(* Logix 5000 project; controller cal1615 1756-L62 rev 16.20; software revision 16.05; part 42 of 78 *)
(* tags used below, declared in another part *)
   AFI : BOOL;   // Always False Bit
   FAULT : BOOL;   // Fault AFI
   p01r02_plc_scan_time_in_sec : REAL;   // System PLC Scan Time in Seconds
   p01r09_pb_global_reset : BOOL;   // System Modes PB: Global Fault Reset
   p20_ao_lo_turret_selected_speed : REAL;   // Letoff Letoff Turret VFD Selected Speed
   p20_di_clutch_prs_ok : BOOL;   // Letoff Modes Accumulator Position Mode
   p20_di_lo_turret : acs800_di_normal;   // Letoff Letoff Turret VFD Drive Inputs
   p20_di_lo_turret_therm : BOOL;   // Letoff Input Letoff Turret Motor Temp Ok
   p20_di_turret_fwd : BOOL;   // Letoff Digital Inputs PB: Turret FWD
   p20_di_turret_pos : BOOL;   // Letoff Digital Inputs PX: Turret in Position
   p20_di_turret_rev : BOOL;   // Letoff Digital Inputs PB: Turret REV
   p20_do_close_nip : BOOL;   // Letoff Digital Output Feedroll Roll Nip Close
   p20_do_wdr_turret : acs800_do_normal;
   p20_param_lo_turret_index_speed : REAL;
   p20_request_run_index_dir : BOOL;   // Letoff Letoff Turret Request Run Index Direction
   p20_request_run_index_rev_dir : BOOL;   // Letoff Letoff Turret Request Run Index Reverse Direction
   p20r01 : routine;   // Letoff Main
   p20r15 : routine;   // Letoff Letoff A VFD
   p20r15_loa_on : BOOL;   // Letoff Letoff A VFD On
   p20r16_lob_on : BOOL;   // Letoff Letoff B On
   p20r18 : routine;   // Letoff Letoff Turret VFD
   p20r18_acc_dec_ramp : SYS_ACC_DEC_RAMP;   // Letoff Letoff Turret VFD Acel Decel Ramp
   p20r18_accel_rate : REAL;
   p20r18_decel_rate : REAL;
   p20r18_index_complete : BOOL;   // Letoff Letoff Turret VFD Index Complete
   p20r18_index_move_timer : TIMER;   // Letoff Letoff Turret VFD Move Timer
   p20r18_index_time : DINT;   // Letoff Letoff Turret Index Time
   p20r18_index_time_offset : DINT;   // Letoff Letoff Turret VFD Index Time Offset (Accel/Decel Rate Difference)
   p20r18_index_timer : TIMER;   // Letoff Letoff Turret Index Timer
   p20r18_pb_index_fwd : BOOL;   // Letoff Letoff Turret VFD PB: Index FWD
   p20r18_pb_index_rev : BOOL;   // Letoff Letoff Turret VFD PB: Index REV
   p20r18_permissive : BOOL;   // Letoff Letoff Turret VFD Permissive
   p20r18_request_index_fwd : BOOL;   // Letoff Letoff Turret Request Index Forward
   p20r18_request_index_rev : BOOL;   // Letoff Letoff Turret Request Index Reverse
   p20r18_selected_speed : REAL;   // Letoff Letoff Turret VFD Selected Speed
   p20r18_timer_fault : TIMER[10];   // Letoff Letoff Turret Fault Dwell Timer
   p20r18_timer_warning : TIMER[4];   // Letoff Letoff Turret VFD Warning Dwell Timer
   p20r18_zero_speed : BOOL;   // Letoff Letoff Turret VFD At Zero Speed
   p21_dint_to_hmi : DINT[16];   // Splice Press
   P21r01 : routine;
   p21r02 : routine;   // Splice Press Misc Control
   p21r02_fault_exists : BOOL;
   p21r02_timer_fault : TIMER[4];   // Splice Press Misc Control Fault Delay
   p21r02_timer_warning : TIMER[4];   // Splice Press Misc Control Warning Delay
   p21r02_unack_fault : BOOL;   // Splice Press Misc Control Unacknowledged Fault Exists
   p21r02_unack_warning : BOOL;   // Splice Press Misc Control Unacknowledged Warning Exists
   p21r02_warning_exists : BOOL;
   p21r03 : routine;   // Splice Press Inputs
   p21r04 : routine;   // Splice Press Outputs
   p21r05 : routine;   // Splice Press Dint to HMI
   p21r06 : routine;   // Splice Press Real to HMI
   p21r07 : routine;   // Splice Press Alarms
   p21r08 : routine;   // Splice Press Warnings
   p21r09 : routine;   // Splice Press Modes
   p21r10 : routine;   // Splice Press Sequence
   p21r16 : routine;   // Splice Press Temperature Control
(* P20_Letoff, continued *)

ROUTINE R18_Letoff_Turret_VFD   (* ladder *)
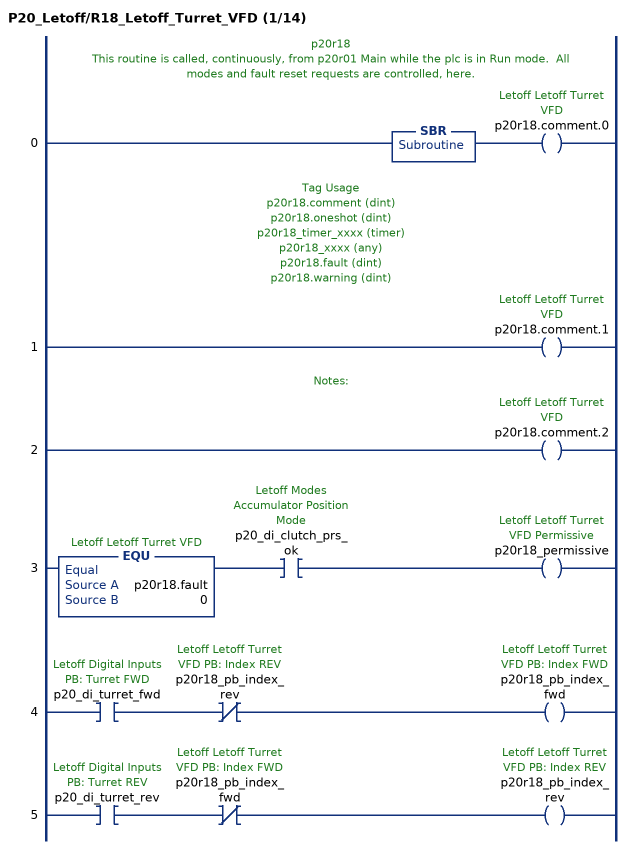
   // p20r18
   // This routine is called, continuously, from p20r01 Main while the plc is in Run mode.  All modes and fault reset requests are controlled, here.
   0: SBR()OTE(p20r18.comment.0);
   // Tag Usage
   // p20r18.comment (dint)
   // p20r18.oneshot (dint)
   // p20r18_timer_xxxx (timer)
   // p20r18_xxxx (any)
   // p20r18.fault (dint)
   // p20r18.warning (dint)
   1: OTE(p20r18.comment.1);
   // Notes:
   2: OTE(p20r18.comment.2);
   3: EQU(p20r18.fault,0)XIC(p20_di_clutch_prs_ok)OTE(p20r18_permissive);
   4: XIC(p20_di_turret_fwd)XIO(p20r18_pb_index_rev)OTE(p20r18_pb_index_fwd);
   5: XIC(p20_di_turret_rev)XIO(p20r18_pb_index_fwd)OTE(p20r18_pb_index_rev);
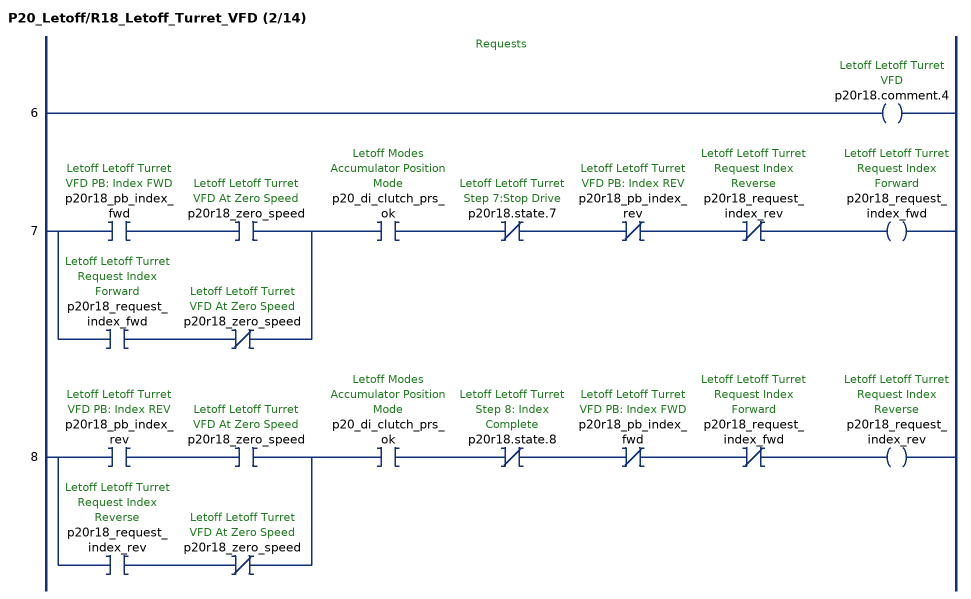
   // Requests
   6: OTE(p20r18.comment.4);
   7: [XIC(p20r18_pb_index_fwd) XIC(p20r18_zero_speed) ,XIC(p20r18_request_index_fwd) XIO(p20r18_zero_speed) ]XIC(p20_di_clutch_prs_ok)XIO(p20r18.state.7)XIO(p20r18_pb_index_rev)XIO(p20r18_request_index_rev)OTE(p20r18_request_index_fwd);
   8: [XIC(p20r18_pb_index_rev) XIC(p20r18_zero_speed) ,XIC(p20r18_request_index_rev) XIO(p20r18_zero_speed) ]XIC(p20_di_clutch_prs_ok)XIO(p20r18.state.8)XIO(p20r18_pb_index_fwd)XIO(p20r18_request_index_fwd)OTE(p20r18_request_index_rev);
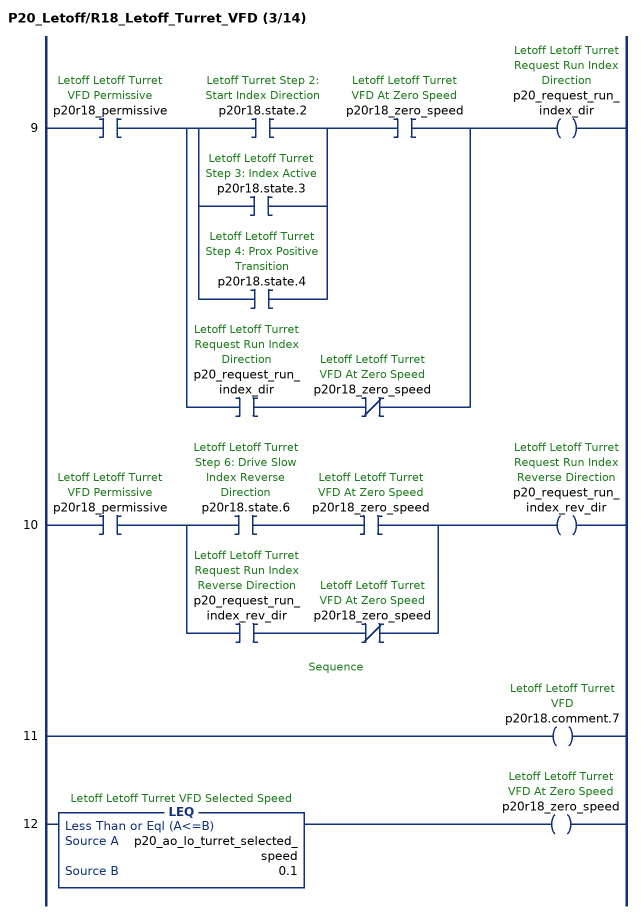
   9: XIC(p20r18_permissive)[[XIC(p20r18.state.2) ,XIC(p20r18.state.3) ,XIC(p20r18.state.4) ] XIC(p20r18_zero_speed) ,XIC(p20_request_run_index_dir) XIO(p20r18_zero_speed) ]OTE(p20_request_run_index_dir);
   10: XIC(p20r18_permissive)[XIC(p20r18.state.6) XIC(p20r18_zero_speed) ,XIC(p20_request_run_index_rev_dir) XIO(p20r18_zero_speed) ]OTE(p20_request_run_index_rev_dir);
   // Sequence
   11: OTE(p20r18.comment.7);
   12: LEQ(p20_ao_lo_turret_selected_speed,0.1)OTE(p20r18_zero_speed);
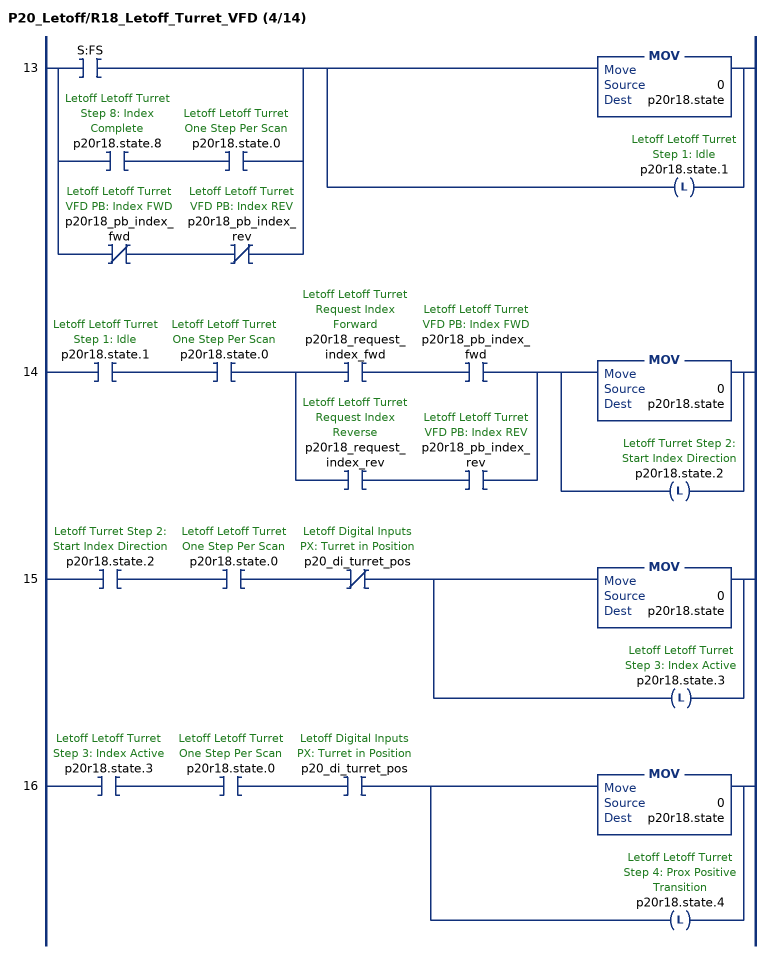
   13: [XIC(S:FS) ,XIC(p20r18.state.8) XIC(p20r18.state.0) ,XIO(p20r18_pb_index_fwd) XIO(p20r18_pb_index_rev) ][MOV(0,p20r18.state) ,OTL(p20r18.state.1) ];
   14: XIC(p20r18.state.1)XIC(p20r18.state.0)[XIC(p20r18_request_index_fwd) XIC(p20r18_pb_index_fwd) ,XIC(p20r18_request_index_rev) XIC(p20r18_pb_index_rev) ][MOV(0,p20r18.state) ,OTL(p20r18.state.2) ];
   15: XIC(p20r18.state.2)XIC(p20r18.state.0)XIO(p20_di_turret_pos)[MOV(0,p20r18.state) ,OTL(p20r18.state.3) ];
   16: XIC(p20r18.state.3)XIC(p20r18.state.0)XIC(p20_di_turret_pos)[MOV(0,p20r18.state) ,OTL(p20r18.state.4) ];
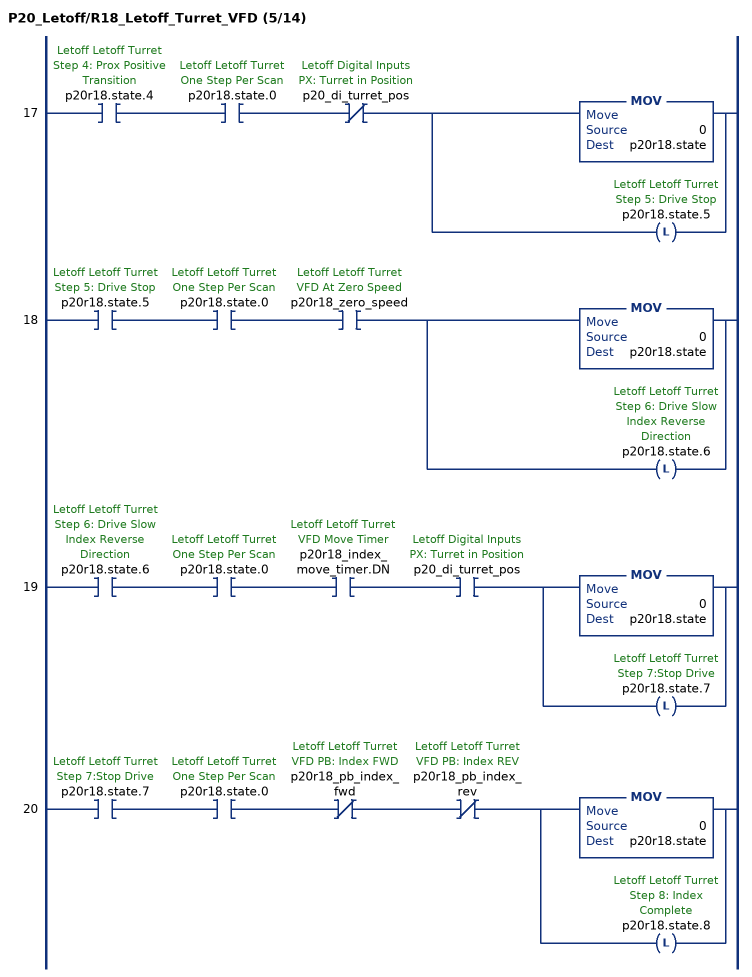
   17: XIC(p20r18.state.4)XIC(p20r18.state.0)XIO(p20_di_turret_pos)[MOV(0,p20r18.state) ,OTL(p20r18.state.5) ];
   18: XIC(p20r18.state.5)XIC(p20r18.state.0)XIC(p20r18_zero_speed)[MOV(0,p20r18.state) ,OTL(p20r18.state.6) ];
   19: XIC(p20r18.state.6)XIC(p20r18.state.0)XIC(p20r18_index_move_timer.DN)XIC(p20_di_turret_pos)[MOV(0,p20r18.state) ,OTL(p20r18.state.7) ];
   20: XIC(p20r18.state.7)XIC(p20r18.state.0)XIO(p20r18_pb_index_fwd)XIO(p20r18_pb_index_rev)[MOV(0,p20r18.state) ,OTL(p20r18.state.8) ];
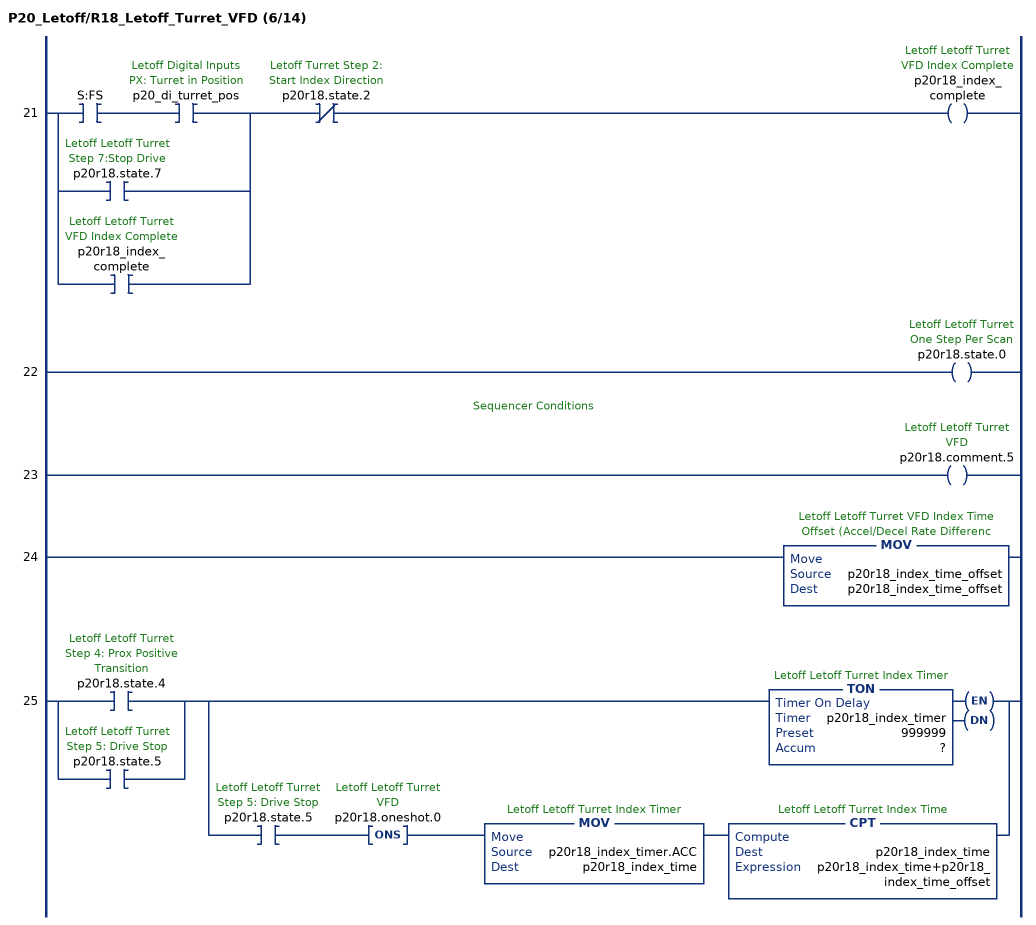
   21: [XIC(S:FS) XIC(p20_di_turret_pos) ,XIC(p20r18.state.7) ,XIC(p20r18_index_complete) ]XIO(p20r18.state.2)OTE(p20r18_index_complete);
   22: OTE(p20r18.state.0);
   // Sequencer Conditions
   23: OTE(p20r18.comment.5);
   24: MOV(p20r18_index_time_offset,p20r18_index_time_offset);
   25: [XIC(p20r18.state.4) ,XIC(p20r18.state.5) ][TON(p20r18_index_timer,?,?) ,XIC(p20r18.state.5) ONS(p20r18.oneshot.0) MOV(p20r18_index_timer.ACC,p20r18_index_time) CPT(p20r18_index_time,p20r18_index_time+p20r18_index_time_offset) ];
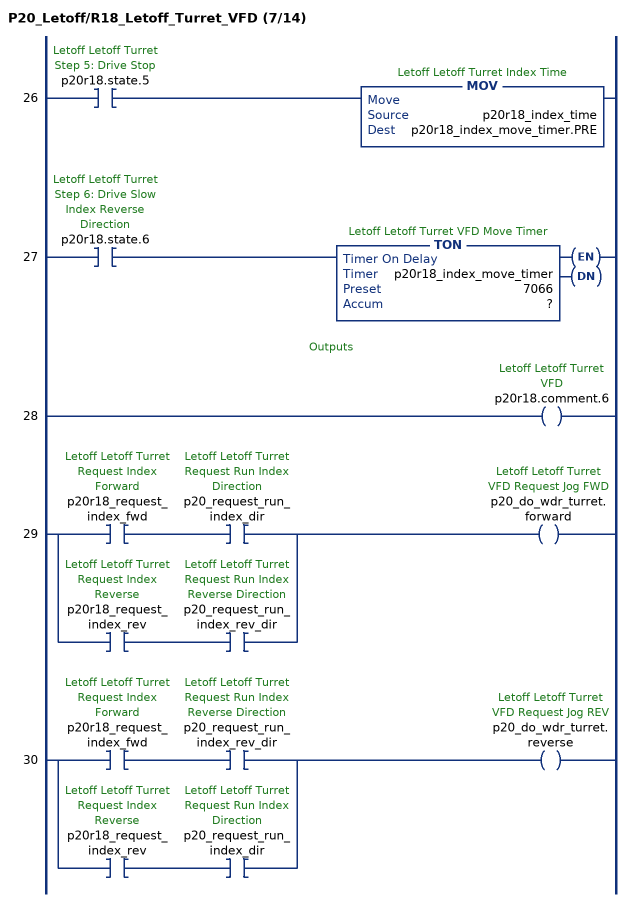
   26: XIC(p20r18.state.5)MOV(p20r18_index_time,p20r18_index_move_timer.PRE);
   27: XIC(p20r18.state.6)TON(p20r18_index_move_timer,?,?);
   // Outputs
   28: OTE(p20r18.comment.6);
   29: [XIC(p20r18_request_index_fwd) XIC(p20_request_run_index_dir) ,XIC(p20r18_request_index_rev) XIC(p20_request_run_index_rev_dir) ]OTE(p20_do_wdr_turret.forward);
   30: [XIC(p20r18_request_index_fwd) XIC(p20_request_run_index_rev_dir) ,XIC(p20r18_request_index_rev) XIC(p20_request_run_index_dir) ]OTE(p20_do_wdr_turret.reverse);
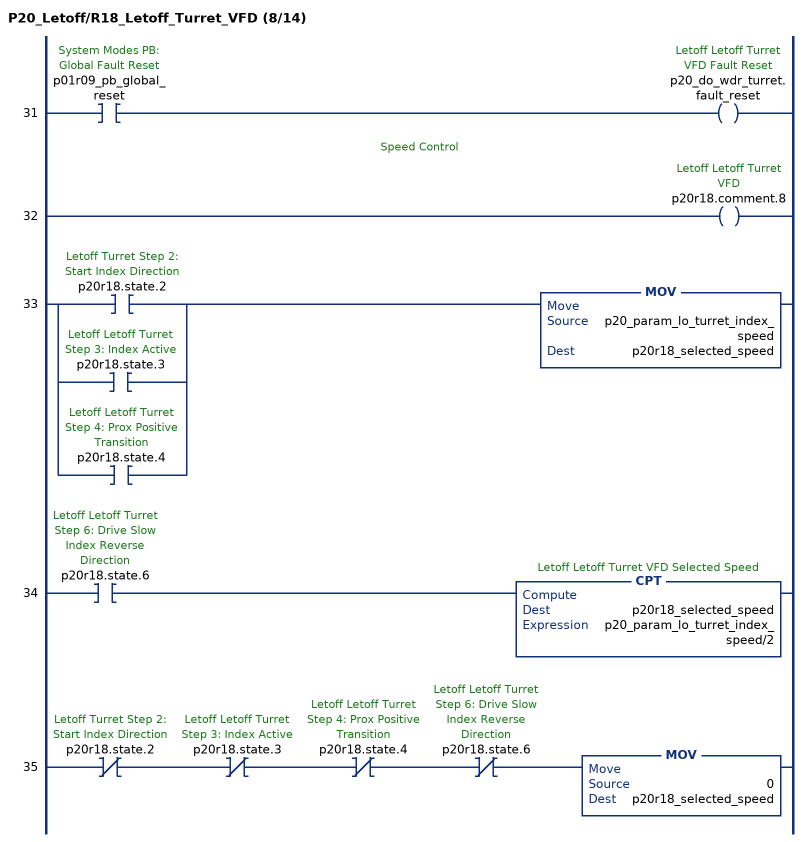
   31: XIC(p01r09_pb_global_reset)OTE(p20_do_wdr_turret.fault_reset);
   // Speed Control
   32: OTE(p20r18.comment.8);
   33: [XIC(p20r18.state.2) ,XIC(p20r18.state.3) ,XIC(p20r18.state.4) ]MOV(p20_param_lo_turret_index_speed,p20r18_selected_speed);
   34: XIC(p20r18.state.6)CPT(p20r18_selected_speed,p20_param_lo_turret_index_speed/2);
   35: XIO(p20r18.state.2)XIO(p20r18.state.3)XIO(p20r18.state.4)XIO(p20r18.state.6)MOV(0,p20r18_selected_speed);
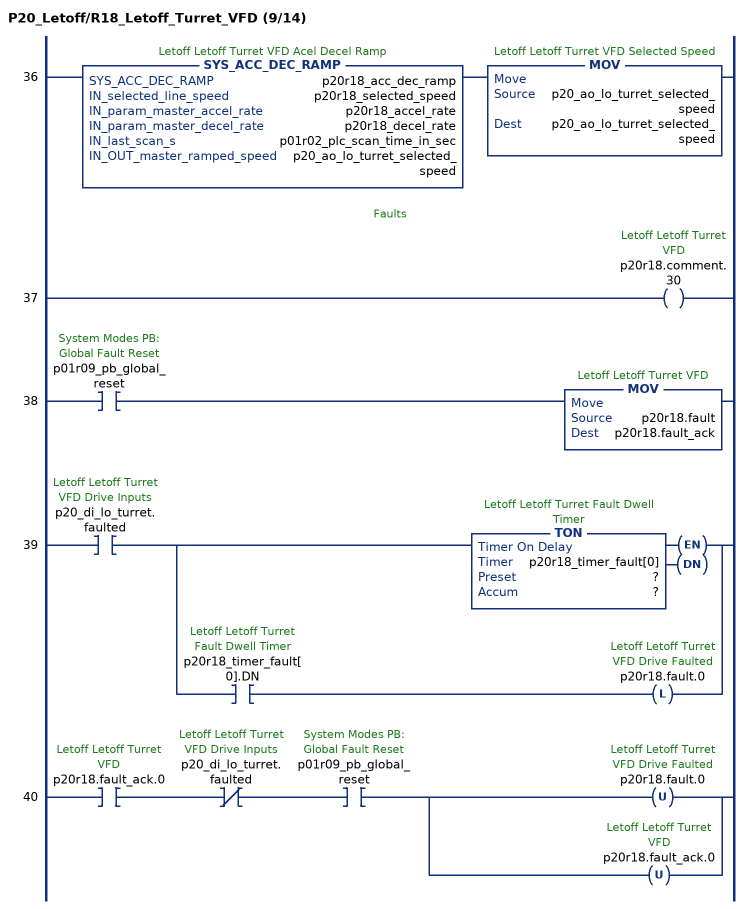
   36: SYS_ACC_DEC_RAMP(p20r18_acc_dec_ramp,p20r18_selected_speed,p20r18_accel_rate,p20r18_decel_rate,p01r02_plc_scan_time_in_sec,p20_ao_lo_turret_selected_speed)MOV(p20_ao_lo_turret_selected_speed,p20_ao_lo_turret_selected_speed);
   // Faults
   37: OTE(p20r18.comment.30);
   38: XIC(p01r09_pb_global_reset)MOV(p20r18.fault,p20r18.fault_ack);
   39: XIC(p20_di_lo_turret.faulted)[TON(p20r18_timer_fault[0],?,?) ,XIC(p20r18_timer_fault[0].DN) OTL(p20r18.fault.0) ];
   40: XIC(p20r18.fault_ack.0)XIO(p20_di_lo_turret.faulted)XIC(p01r09_pb_global_reset)[OTU(p20r18.fault.0) ,OTU(p20r18.fault_ack.0) ];
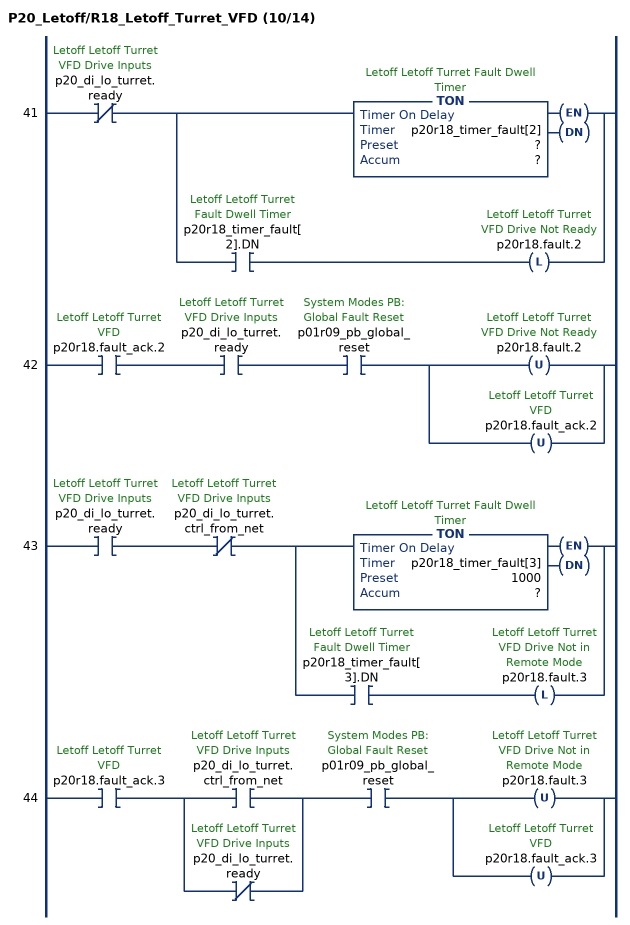
   41: XIO(p20_di_lo_turret.ready)[TON(p20r18_timer_fault[2],?,?) ,XIC(p20r18_timer_fault[2].DN) OTL(p20r18.fault.2) ];
   42: XIC(p20r18.fault_ack.2)XIC(p20_di_lo_turret.ready)XIC(p01r09_pb_global_reset)[OTU(p20r18.fault.2) ,OTU(p20r18.fault_ack.2) ];
   43: XIC(p20_di_lo_turret.ready)XIO(p20_di_lo_turret.ctrl_from_net)[TON(p20r18_timer_fault[3],?,?) ,XIC(p20r18_timer_fault[3].DN) OTL(p20r18.fault.3) ];
   44: XIC(p20r18.fault_ack.3)[XIC(p20_di_lo_turret.ctrl_from_net) ,XIO(p20_di_lo_turret.ready) ]XIC(p01r09_pb_global_reset)[OTU(p20r18.fault.3) ,OTU(p20r18.fault_ack.3) ];
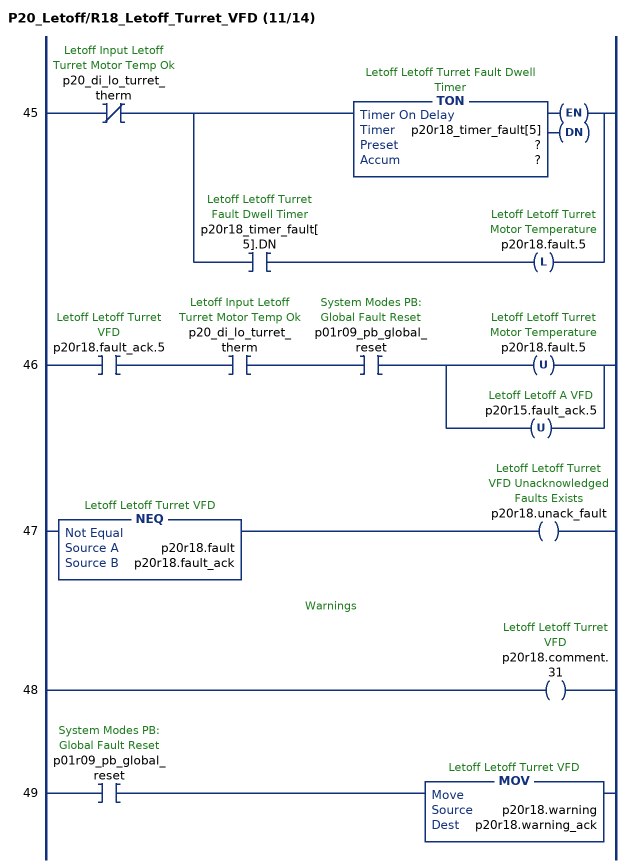
   45: XIO(p20_di_lo_turret_therm)[TON(p20r18_timer_fault[5],?,?) ,XIC(p20r18_timer_fault[5].DN) OTL(p20r18.fault.5) ];
   46: XIC(p20r18.fault_ack.5)XIC(p20_di_lo_turret_therm)XIC(p01r09_pb_global_reset)[OTU(p20r18.fault.5) ,OTU(p20r15.fault_ack.5) ];
   47: NEQ(p20r18.fault,p20r18.fault_ack)OTE(p20r18.unack_fault);
   // Warnings
   48: OTE(p20r18.comment.31);
   49: XIC(p01r09_pb_global_reset)MOV(p20r18.warning,p20r18.warning_ack);
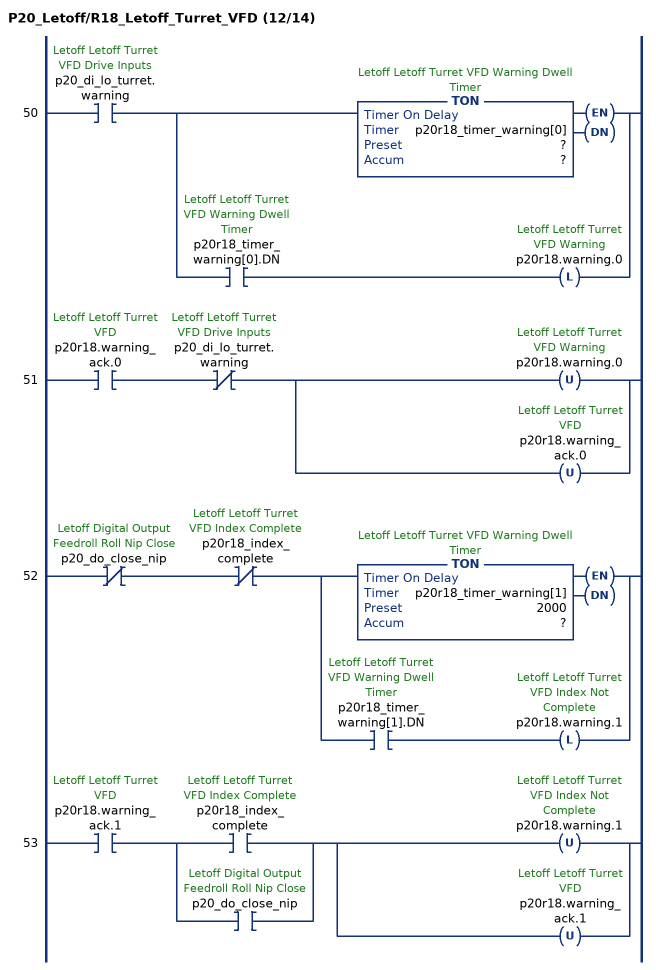
   50: XIC(p20_di_lo_turret.warning)[TON(p20r18_timer_warning[0],?,?) ,XIC(p20r18_timer_warning[0].DN) OTL(p20r18.warning.0) ];
   51: XIC(p20r18.warning_ack.0)XIO(p20_di_lo_turret.warning)[OTU(p20r18.warning.0) ,OTU(p20r18.warning_ack.0) ];
   52: XIO(p20_do_close_nip)XIO(p20r18_index_complete)[TON(p20r18_timer_warning[1],?,?) ,XIC(p20r18_timer_warning[1].DN) OTL(p20r18.warning.1) ];
   53: XIC(p20r18.warning_ack.1)[XIC(p20r18_index_complete) ,XIC(p20_do_close_nip) ][OTU(p20r18.warning.1) ,OTU(p20r18.warning_ack.1) ];
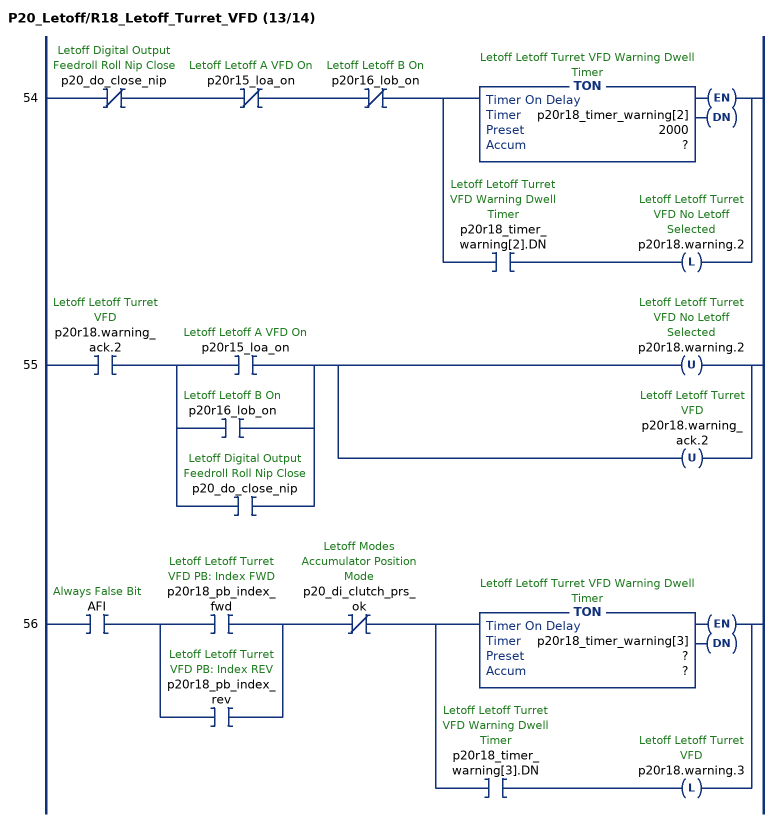
   54: XIO(p20_do_close_nip)XIO(p20r15_loa_on)XIO(p20r16_lob_on)[TON(p20r18_timer_warning[2],?,?) ,XIC(p20r18_timer_warning[2].DN) OTL(p20r18.warning.2) ];
   55: XIC(p20r18.warning_ack.2)[XIC(p20r15_loa_on) ,XIC(p20r16_lob_on) ,XIC(p20_do_close_nip) ][OTU(p20r18.warning.2) ,OTU(p20r18.warning_ack.2) ];
   56: XIC(AFI)[XIC(p20r18_pb_index_fwd) ,XIC(p20r18_pb_index_rev) ]XIO(p20_di_clutch_prs_ok)[TON(p20r18_timer_warning[3],?,?) ,XIC(p20r18_timer_warning[3].DN) OTL(p20r18.warning.3) ];
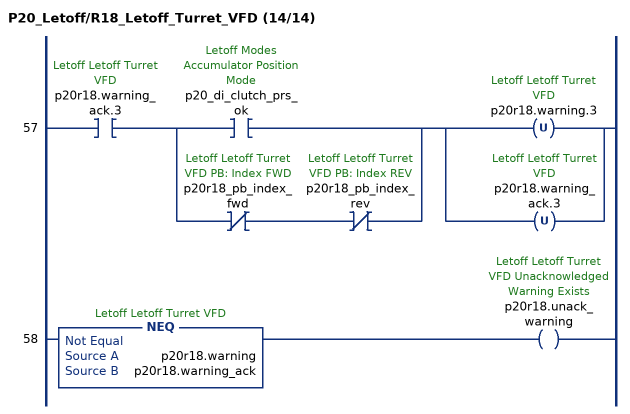
   57: XIC(p20r18.warning_ack.3)[XIC(p20_di_clutch_prs_ok) ,XIO(p20r18_pb_index_fwd) XIO(p20r18_pb_index_rev) ][OTU(p20r18.warning.3) ,OTU(p20r18.warning_ack.3) ];
   58: NEQ(p20r18.warning,p20r18.warning_ack)OTE(p20r18.unack_warning);
END_ROUTINE
END_PROGRAM

PROGRAM P21_Splice_Press   (* main routine R01_Main *)

ROUTINE R01_Main   (* ladder *)
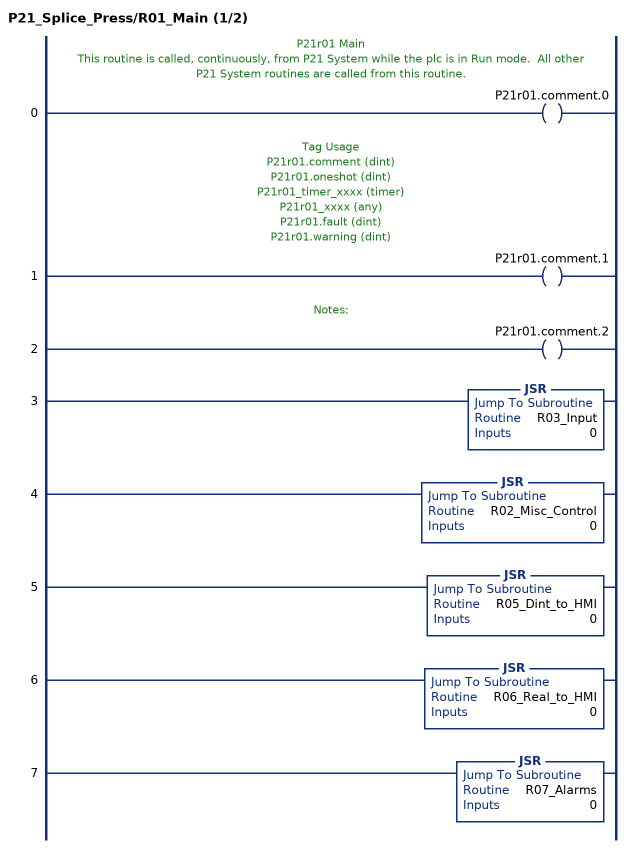
   // P21r01 Main
   // This routine is called, continuously, from P21 System while the plc is in Run mode.  All other P21 System routines are called from this routine.
   0: OTE(P21r01.comment.0);
   // Tag Usage
   // P21r01.comment (dint)
   // P21r01.oneshot (dint)
   // P21r01_timer_xxxx (timer)
   // P21r01_xxxx (any)
   // P21r01.fault (dint)
   // P21r01.warning (dint)
   1: OTE(P21r01.comment.1);
   // Notes:
   2: OTE(P21r01.comment.2);
   3: JSR(R03_Input,0);
   4: JSR(R02_Misc_Control,0);
   5: JSR(R05_Dint_to_HMI,0);
   6: JSR(R06_Real_to_HMI,0);
   7: JSR(R07_Alarms,0);
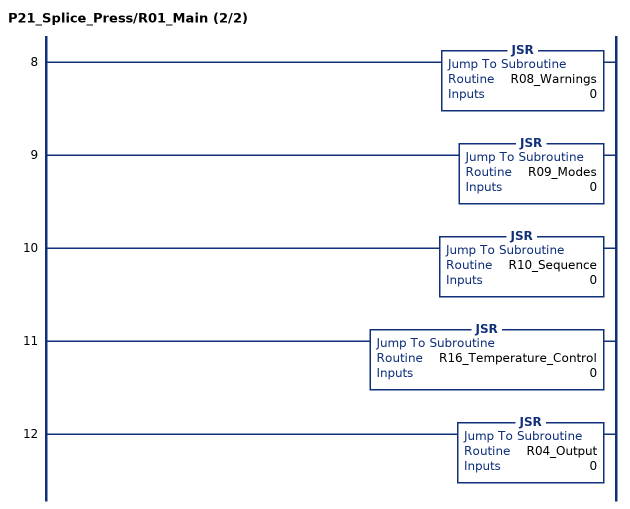
   8: JSR(R08_Warnings,0);
   9: JSR(R09_Modes,0);
   10: JSR(R10_Sequence,0);
   11: JSR(R16_Temperature_Control,0);
   12: JSR(R04_Output,0);
END_ROUTINE

ROUTINE R02_Misc_Control   (* ladder *)
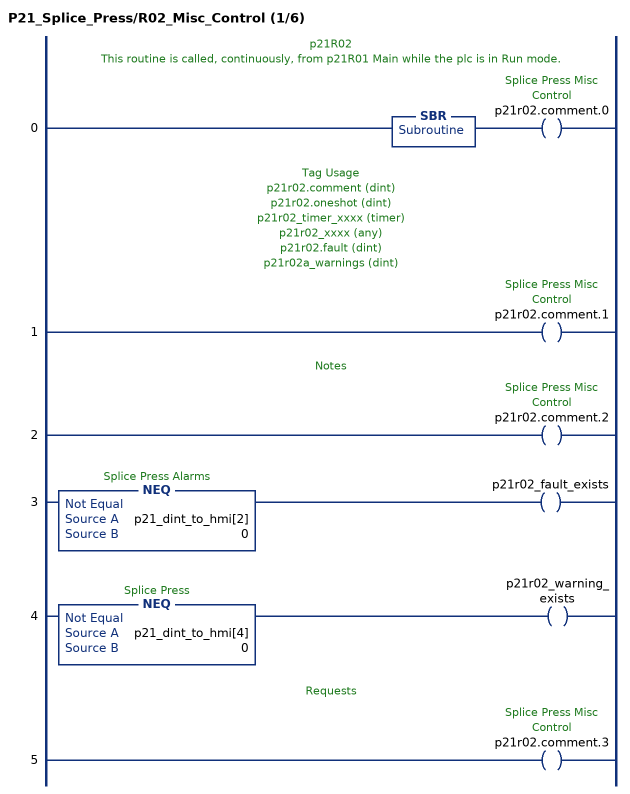
   // p21R02
   // This routine is called, continuously, from p21R01 Main while the plc is in Run mode.
   0: SBR()OTE(p21r02.comment.0);
   // Tag Usage
   // p21r02.comment (dint)
   // p21r02.oneshot (dint)
   // p21r02_timer_xxxx (timer)
   // p21r02_xxxx (any)
   // p21r02.fault (dint)
   // p21r02a_warnings (dint)
   1: OTE(p21r02.comment.1);
   // Notes
   2: OTE(p21r02.comment.2);
   3: NEQ(p21_dint_to_hmi[2],0)OTE(p21r02_fault_exists);
   4: NEQ(p21_dint_to_hmi[4],0)OTE(p21r02_warning_exists);
   // Requests
   5: OTE(p21r02.comment.3);
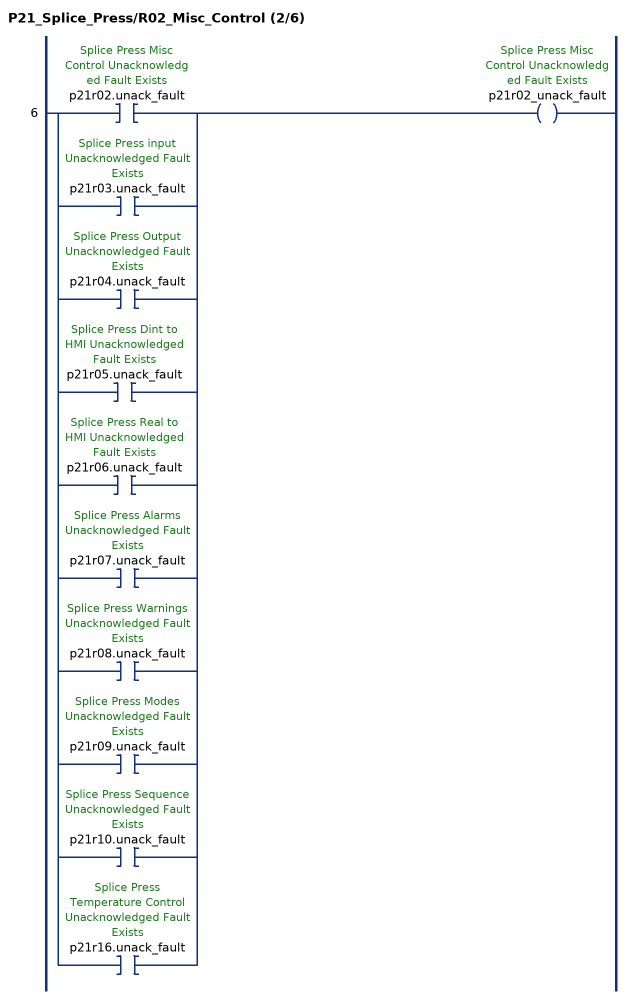
   6: [XIC(p21r02.unack_fault) ,XIC(p21r03.unack_fault) ,XIC(p21r04.unack_fault) ,XIC(p21r05.unack_fault) ,XIC(p21r06.unack_fault) ,XIC(p21r07.unack_fault) ,XIC(p21r08.unack_fault) ,XIC(p21r09.unack_fault) ,XIC(p21r10.unack_fault) ,XIC(p21r16.unack_fault) ]OTE(p21r02_unack_fault);
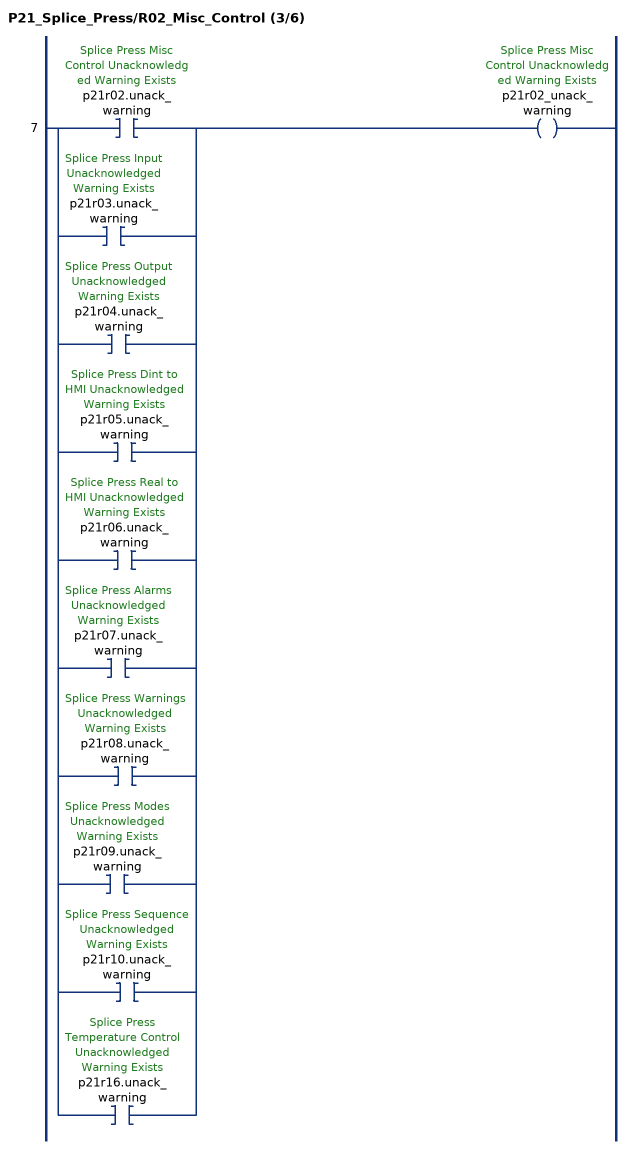
   7: [XIC(p21r02.unack_warning) ,XIC(p21r03.unack_warning) ,XIC(p21r04.unack_warning) ,XIC(p21r05.unack_warning) ,XIC(p21r06.unack_warning) ,XIC(p21r07.unack_warning) ,XIC(p21r08.unack_warning) ,XIC(p21r09.unack_warning) ,XIC(p21r10.unack_warning) ,XIC(p21r16.unack_warning) ]OTE(p21r02_unack_warning);
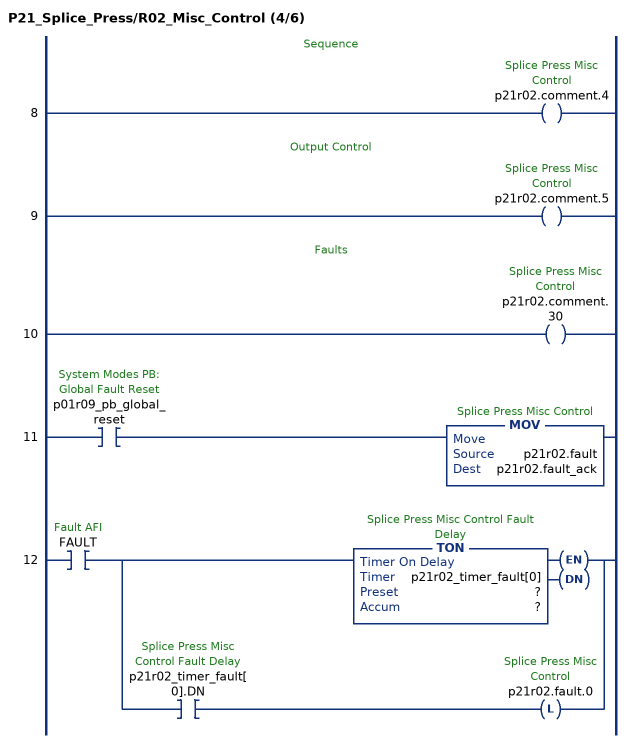
   // Sequence
   8: OTE(p21r02.comment.4);
   // Output Control
   9: OTE(p21r02.comment.5);
   // Faults
   10: OTE(p21r02.comment.30);
   11: XIC(p01r09_pb_global_reset)MOV(p21r02.fault,p21r02.fault_ack);
   12: XIC(FAULT)[TON(p21r02_timer_fault[0],?,?) ,XIC(p21r02_timer_fault[0].DN) OTL(p21r02.fault.0) ];
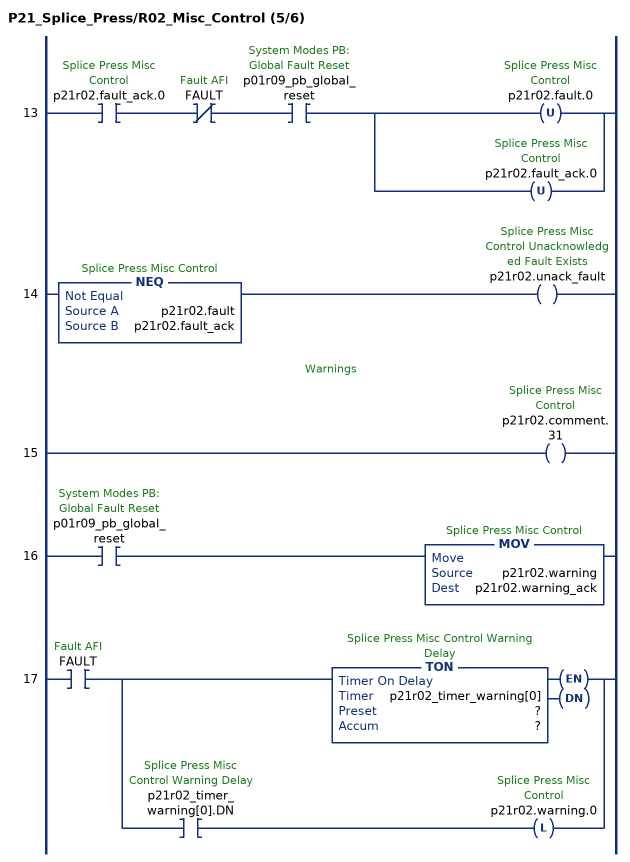
   13: XIC(p21r02.fault_ack.0)XIO(FAULT)XIC(p01r09_pb_global_reset)[OTU(p21r02.fault.0) ,OTU(p21r02.fault_ack.0) ];
   14: NEQ(p21r02.fault,p21r02.fault_ack)OTE(p21r02.unack_fault);
   // Warnings
   15: OTE(p21r02.comment.31);
   16: XIC(p01r09_pb_global_reset)MOV(p21r02.warning,p21r02.warning_ack);
   17: XIC(FAULT)[TON(p21r02_timer_warning[0],?,?) ,XIC(p21r02_timer_warning[0].DN) OTL(p21r02.warning.0) ];
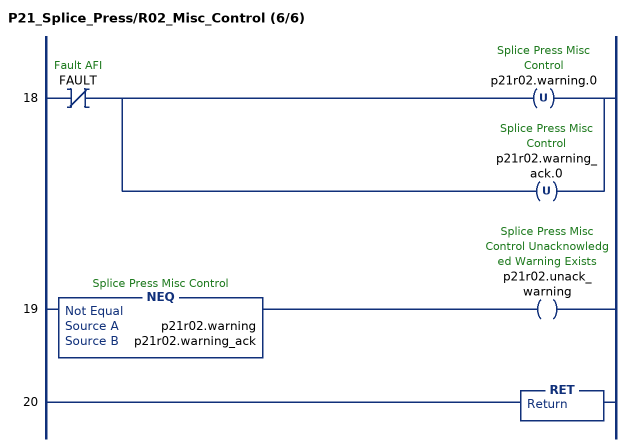
   18: XIO(FAULT)[OTU(p21r02.warning.0) ,OTU(p21r02.warning_ack.0) ];
   19: NEQ(p21r02.warning,p21r02.warning_ack)OTE(p21r02.unack_warning);
   20: RET();
END_ROUTINE
